# B&R Automation Studio project lab_2
Automation Studio 4.5.2.102

## Configuration lab_config

CPU 4PP065.0571-P74, AutomationRuntime D4.52, Build 4.1.2, Vc V4.52.0, Safety 1.6

### Task classes (Cpu.sw)
```
Cyclic#1 (cycle 2000 us, tolerance 0 us):
  ncsdcctrl <- ncsdcctrl.prg
Cyclic#8:
  Program1 <- Program1.prg
NcDataObjects: acp10etxen <- acp10etxen.dob, gAxis01a <- gAxis01obj.gAxis01a.dob, gAxis01i <- gAxis01obj.gAxis01i.dob, gAxis02a <- gAxis02obj.gAxis02a.dob, gAxis02i <- gAxis02obj.gAxis02i.dob
VcDataObjects: Visu <- Visu.dob
Binaries: vcpdsw, udbdef, vcrt, vcpfmtcx, Visu03, vcfile, vcgclass, arial, vcdsint, vcmgr, vcdsloc, vcfntttf, Visu02, vccovl, vcshared, arialbd, vcalarm, vcptelo, vcpdpp30, vccbtn, Visu01, vccnum, vcbclass, vcpfpp30, vctcal, TCData, iomap, asfw, Role, ashwac, sysconf, ashwd, User, arconfig, acp10cfg, Acp10map, vcctext
Libraries: Acp10man, Acp10par, NcGlobal, Acp10sdc, AsBrStr, Acp10_MC, brsystem, sys_lib, runtime, Library1, vcresman, asieccon, fileio, astime, dataobj, powerlnk
```

### Hardware
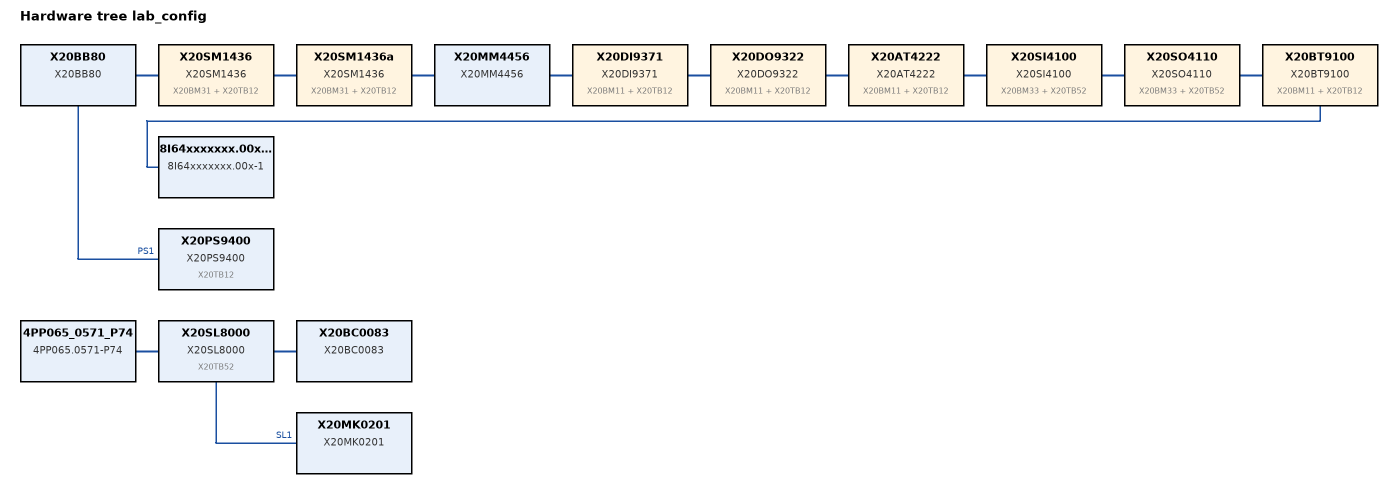
```
4PP065_0571_P74 : 4PP065.0571-P74 v1.1.2.0
  Connector IF5:
    ActivateDevice = 1
    Mode = Manual
    InternetAddress = 10.0.1.10
    SubnetMask = 255.255.255.0
  ConfigurationID = labBR
  Simulation = 1
  TimerDeviceType = EPLX2X
  TimerDevice = 4PP065_0571_P74.IF4
  TaskClassIdleTime = 2000
  Cyclic1Duration = 2000
  Cyclic1Tolerance = 0
  Cyclic1Output = 1
  VcObjectName = Visu
8I64xxxxxxx.00x-1a : 8I64xxxxxxx.00x-1 v1.3.9.1  [X2X1 -> X20BT9100.X2X1 [Cable Type=X2XCable, Length=10, Version=1.0.0.2]]
  packedETAD = packed
  packedETI = packed
  packedCMDD = packed
  packedCMI = packed
  UNS = 220
  NCR = 10
  NSP = 890
  COS = 64
  RSC = 33000
X20AT4222 : X20AT4222 v1.2.3.0  [SS1 -> X20TB12d.SS; SL -> X20BM11b.SL1]
X20BB80 : X20BB80 v1.0.2.0
X20BC0083 : X20BC0083 v2.7.0.0  [PLK1 -> X20SL8000.PLK2 [Cable Type=PowerlinkCable, Length=10, Version=1.0.0.2]; SL -> X20BB80.SL1]
X20BM11 : X20BM11 v1.0.0.1  [X2X1 -> X20MM4456.X2X2]
X20BM11a : X20BM11 v1.0.0.1  [X2X1 -> X20BM11.X2X2]
X20BM11b : X20BM11 v1.0.0.1  [X2X1 -> X20BM11a.X2X2]
X20BM11c : X20BM11 v1.0.0.1  [X2X1 -> X20BM33a.X2X2]
X20BM31 : X20BM31 v1.0.0.1  [X2X1 -> X20BB80.IF1]
X20BM31a : X20BM31 v1.0.0.1  [X2X1 -> X20BM31.X2X2]
X20BM33 : X20BM33 v1.0.0.4  [X2X1 -> X20BM11b.X2X2]
X20BM33a : X20BM33 v1.0.0.4  [X2X1 -> X20BM33.X2X2]
X20BT9100 : X20BT9100 v1.0.3.0  [SS1 -> X20TB12e.SS; SL -> X20BM11c.SL1]
X20DI9371 : X20DI9371 v1.0.2.0  [SS1 -> X20TB12b.SS; SL -> X20BM11.SL1]
X20DO9322 : X20DO9322 v1.0.3.0  [SS1 -> X20TB12c.SS; SL -> X20BM11a.SL1]
X20MK0201 : X20MK0201 v1.0.0.0  [SL -> X20SL8000.SL1]
X20MM4456 : X20MM4456 v1.1.5.0  [X2X1 -> X20BM31a.X2X2]
X20PS9400 : X20PS9400 v1.0.2.4  [SS1 -> X20TB12.SS; PS -> X20BB80.PS1]
X20SI4100 : X20SI4100 v1.10.1.1  [SS1 -> X20TB52a.SS; SL -> X20BM33.SL1]
X20SL8000 : X20SL8000 v1.6.5.1  [PLK1 -> 4PP065_0571_P74.IF4 [Cable Type=PowerlinkCable, Length=10, Version=1.0.0.2]; PLK2 -> X20BC0083.PLK1 [Cable Type=PowerlinkCable, Length=10, Version=1.0.0.2]; SS1 -> X20TB52.SS]
  SafeProject = SafeLOGIC-1
X20SM1436 : X20SM1436 v1.4.2.1  [SS1 -> X20TB12a.SS; SL -> X20BM31.SL1]
X20SM1436a : X20SM1436 v1.4.2.1  [SS1 -> X20TB12f.SS; SL -> X20BM31a.SL1]
X20SO4110 : X20SO4110 v1.10.1.1  [SS1 -> X20TB52b.SS; SL -> X20BM33a.SL1]
  SafeModuleID = 3
X20TB12 : X20TB12 v1.0.0.0
X20TB12a : X20TB12 v1.0.0.0
X20TB12b : X20TB12 v1.0.0.0
X20TB12c : X20TB12 v1.0.0.0
X20TB12d : X20TB12 v1.0.0.0
X20TB12e : X20TB12 v1.0.0.0
X20TB12f : X20TB12 v1.0.0.0
X20TB52 : X20TB52 v1.0.0.1
X20TB52a : X20TB52 v1.0.0.1
X20TB52b : X20TB52 v1.0.0.1
```

### IoMap.iom - 4PP065_0571_P74/IoMap.iom
```iecst
VAR_CONFIG
	::driveSM.STATE AT %IW."8I64xxxxxxx.00x-1a".ETAD_Input;
	::driveSM.CMD AT %QW."8I64xxxxxxx.00x-1a".CMDD_Output;
	Cyclic#1.gAxis02_DrvIf.iLifeCnt AT %IB."8I64xxxxxxx.00x-1a".SDC_LifeCnt;
	Cyclic#1.gAxis02_DrvIf.iDrvOK AT %IX."8I64xxxxxxx.00x-1a".ETAD_Input_Bool_02;
	Cyclic#1.gAxis02_DrvIf.oSetTime AT %QW."8I64xxxxxxx.00x-1a".SDC_SetTime;
	Cyclic#1.::driveSM.speed AT %QW."8I64xxxxxxx.00x-1a".LFRD_Output;
	Cyclic#1.gAxis02_DiDoIf.iLifeCntDriveReady AT %IB."8I64xxxxxxx.00x-1a".SDC_LifeCnt;
	Cyclic#1.gAxis02_DiDoIf.iLifeCntDriveEnable AT %IB."8I64xxxxxxx.00x-1a".SDC_LifeCnt;
	Cyclic#1.gAxis02_DiDoIf.oDriveEnable AT %QX."8I64xxxxxxx.00x-1a".CMDD_Output_Bool_00;
	Cyclic#1.gAxis02_ModuleOk AT %QX."8I64xxxxxxx.00x-1a".CMDD_Output_Bool_01;
	Cyclic#1.gAxis02_ModuleOk AT %QX."8I64xxxxxxx.00x-1a".CMDD_Output_Bool_02;
	Cyclic#1.gAxis02_ModuleOk AT %IX."8I64xxxxxxx.00x-1a".ModuleOk;
	Cyclic#1.gAxis02_DiDoIf.oDriveEnable AT %QX."8I64xxxxxxx.00x-1a".CMDD_Output_Bool_03;
	Cyclic#1.gAxis02_DiDoIf.iDriveReady AT %IX."8I64xxxxxxx.00x-1a".ETAD_Input_Bool_02;
	::DoorSM.direction AT %IX."X20DI9371".DigitalInput01;
	::DoorSM.s0 AT %IX."X20DI9371".DigitalInput02;
	::DoorSM.s1 AT %IX."X20DI9371".DigitalInput03;
	::DoorSM.s2 AT %IX."X20DI9371".DigitalInput04;
	::DoorSM.s3 AT %IX."X20DI9371".DigitalInput05;
	::ledSM.led1 AT %QX."X20DO9322".DigitalOutput02;
	::ledSM.led2 AT %QX."X20DO9322".DigitalOutput03;
	::ledSM.led3 AT %QX."X20DO9322".DigitalOutput04;
	::ledSM.led4 AT %QX."X20DO9322".DigitalOutput05;
END_VAR
```

### Acp10map.ncm - 4PP065_0571_P74/Motion/Acp10map.ncm
```
NcMapping (NcSwId=Acp10)
  NcObject X20SM1436_ncAXIS1 (ModuleId=X20SM1436, ModuleAddress=SDC_IF1.ST1, Type=ncAXIS, Channel=1, AcoposSimulation=Off, Disabled=TRUE, ModuleDisabled=FALSE)
  NcObject X20SM1436a_ncAXIS1 (ModuleId=X20SM1436a, ModuleAddress=SDC_IF1.ST2, Type=ncAXIS, Channel=1, AcoposSimulation=Off, Disabled=TRUE, ModuleDisabled=FALSE)
  NcObject gAxis02 (ModuleId=8I64xxxxxxx.00x-1a, ModuleAddress=SDC_IF1.ST3, Type=ncAXIS, Channel=1, AcoposSimulation=Off, InitParameter=gAxis02i, AcoposParameter=gAxis02a, Disabled=FALSE, ModuleDisabled=FALSE)
```

## Logical view

### Global.var - Global variables
```iecst
VAR
	DoorSM : DoorStateMachine;
	speed : INT := 500;
	gAxis01 : ACP10AXIS_typ;
	gAxis01_HW : SdcHwCfg_typ := (0);
	gAxis01_DrvIf : SdcDrvIf16_typ := (0);
	gAxis01_DiDoIf : SdcDiDoIf_typ := (0);
	gAxis01_ModuleOk : BOOL := 0;
	gAxis02 : ACP10AXIS_typ;
	gAxis02_HW : SdcHwCfg_typ := (0);
	gAxis02_DrvIf : SdcDrvIf16_typ := (0);
	gAxis02_DiDoIf : SdcDiDoIf_typ := (0);
	gAxis02_ModuleOk : BOOL := 0;
	ledSM : LedStateMachine;
	driveSM : DriveStateMachine;
END_VAR
```

- Visualisation Logical/Visu (not shown)

### Program Logical/Program1 (ANSIC)

#### Cyclic.c
```c
#include <bur/plctypes.h>

#ifdef _DEFAULT_INCLUDES
	#include <AsDefault.h>
#endif

void _CYCLIC ProgramCyclic(void)
{

	DoorStateMachine(&DoorSM);
	driveSM.speed = DoorSM.speed;
	DriveStateMachine(&driveSM);
	ledSM.state = DoorSM.state;
	LedStateMachine(&ledSM);
}
```

#### Init.c
```c
#include <bur/plctypes.h>

#ifdef _DEFAULT_INCLUDES
	#include <AsDefault.h>
#endif

void _INIT ProgramInit(void)
{
		driveSM.ENABLE = 1;
}
```

### Library Logical/Library1 (ANSIC)

#### Types.typ - Exported data types
```iecst
TYPE
	DoorStates :
		(
		SM_INIT,
		SM_UNKNOWN,
		SM_CLOSE,
		SM_NEG,
		SM_ACC_NEG,
		SM_DEC_NEG,
		SM_OPEN,
		SM_POS,
		SM_ACC_POS,
		SM_DEC_POS
		);
	driveCommands :
		(
		CMD_SWITCHED_ON := 7,
		CMD_DISABLE_VOLTAGE := 0,
		CMD_ENABLED := 15,
		CMD_SHUTDOWN := 6,
		STATE_READY := 33,
		STATE_DISABLED := 64,
		STATE_SWITCHED_ON := 35
		);
END_TYPE
```

#### Library1.fun - Exported functions and function blocks
```iecst
{REDUND_ERROR} FUNCTION_BLOCK LedStateMachine (*TODO: Add your comment here*) (*$GROUP=User,$CAT=User,$GROUPICON=User.png,$CATICON=User.png*)
	VAR_INPUT
		state : UINT;
	END_VAR
	VAR_OUTPUT
		led1 : BOOL;
		led2 : BOOL;
		led3 : BOOL;
		led4 : BOOL;
		timer : INT;
	END_VAR
END_FUNCTION_BLOCK

{REDUND_ERROR} FUNCTION_BLOCK DoorStateMachine (*TODO: Add your comment here*) (*$GROUP=User,$CAT=User,$GROUPICON=User.png,$CATICON=User.png*)
	VAR_INPUT
		state : UINT;
		s0 : BOOL;
		s1 : BOOL;
		s2 : BOOL;
		s3 : BOOL;
		direction : BOOL;
	END_VAR
	VAR_OUTPUT
		speed : INT;
	END_VAR
END_FUNCTION_BLOCK

{REDUND_ERROR} FUNCTION_BLOCK DriveStateMachine (*TODO: Add your comment here*) (*$GROUP=User,$CAT=User,$GROUPICON=User.png,$CATICON=User.png*)
	VAR_INPUT
		STATE : UINT;
		ENABLE : BOOL;
	END_VAR
	VAR_OUTPUT
		CMD : UINT;
		speed : INT;
	END_VAR
END_FUNCTION_BLOCK
```

#### LedStateMachine.c
```c
#include <bur/plctypes.h>
#ifdef __cplusplus
	extern "C"
	{
#endif
	#include "Library1.h"
#ifdef __cplusplus
	};
#endif
/* TODO: Add your comment here */
void LedStateMachine(struct LedStateMachine* inst)
{
	/*TODO: Add your code here*/

	switch(inst->state)
	{
		case SM_INIT:
			{

				break;
			}

		case SM_UNKNOWN:
			{
				if(inst->timer%10==0)
				{
					inst->led1=!inst->led1;
					inst->led2=!inst->led2;
					inst->led3=!inst->led3;
					inst->led4=!inst->led4;
				}
				break;
			}

		case SM_CLOSE:
			{
				inst->led1=1;
				inst->led2=1;
				inst->led3=1;
				inst->led4=1;
				break;
			}
		case SM_NEG:
			{
				inst->led1=0;
				inst->led2=0;
				inst->led3=1;
				inst->led4=1;
				break;
			}
		case SM_ACC_NEG:
			{
				inst->led1=0;
				inst->led2=0;
				inst->led3=0;
				inst->led4=1;
				break;
			}
		case SM_DEC_NEG:
			{
				inst->led1=0;
				inst->led2=1;
				inst->led3=1;
				inst->led4=1;
				break;
			}

		case SM_OPEN:
			{
				inst->led1=0;
				inst->led2=0;
				inst->led3=0;
				inst->led4=0;
				break;
			}
		case SM_POS:
			{
				inst->led1=0;
				inst->led2=0;
				inst->led3=1;
				inst->led4=1;
				break;
			}
		case SM_ACC_POS:
			{
				inst->led1=0;
				inst->led2=1;
				inst->led3=1;
				inst->led4=1;
				break;
			}
		case SM_DEC_POS:
			{
				inst->led1=0;
				inst->led2=0;
				inst->led3=0;
				inst->led4=1;
				break;
			}
	}
	inst->timer++;
}
```

#### DoorStateMachine.c
```c
#include <bur/plctypes.h>
#ifdef __cplusplus
	extern "C"
	{
#endif
	#include "Library1.h"
#ifdef __cplusplus
	};
#endif
/* TODO: Add your comment here */
void DoorStateMachine(struct DoorStateMachine* inst)
{
	/*TODO: Add your code here*/
	switch (inst->state)
	{
		case SM_INIT:
			{
				if(inst->s0==0 && inst->s1==0 && inst->s2==0 && inst->s3==0)
					inst->state=SM_UNKNOWN;
				break;
			}
		case SM_UNKNOWN:
			{
				if (inst->s0 == 1)
					inst->state=SM_CLOSE;
				if (inst->s1 == 1)
					inst->state=SM_ACC_POS;
				if (inst->s2 == 1)
					inst->state=SM_DEC_POS;
				if (inst->s3 == 1)
					inst->state=SM_OPEN;
				break;
			}
		case SM_CLOSE:
			{
				inst->speed = 0;
				if(inst->direction==1)
					inst->state=SM_ACC_POS;
				break;
			}
		case SM_ACC_NEG:
			{
				inst->speed = -200;
				if(inst->direction==1)
					inst->state=SM_DEC_POS;
				if(inst->direction==0 && inst->s2==1)
					inst->state=SM_NEG;
				break;
			}
		case SM_NEG:
			{
				inst->speed = -700;
				if(inst->direction==1)
					inst->state=SM_POS;
				if(inst->direction==0 && inst->s1==1)
					inst->state=SM_DEC_NEG;
				break;

			}

		case SM_DEC_NEG:
			{
				inst->speed = -200;
				if(inst->direction==1)
					inst->state=SM_ACC_POS;
				if(inst->direction==0 && inst->s0==1)
					inst->state=SM_CLOSE;
				break;
			}
		case SM_OPEN:
			{
				inst->speed = 0;
				if(inst->direction==0)
					inst->state=SM_ACC_NEG;
				break;
			}
		case SM_ACC_POS:
			{
				inst->speed = 200;
				if(inst->direction==0)
					inst->state=SM_DEC_NEG;
				if(inst->direction==1 && inst->s1==1)
					inst->state=SM_POS;
				break;
			}
		case SM_POS:
			{
				inst->speed = 700;
				if(inst->direction==0)
					inst->state=SM_NEG;
				if(inst->direction==1 && inst->s2==1)
					inst->state=SM_DEC_POS;
				break;
			}

		case SM_DEC_POS:
			{
				inst->speed = 200;
				if(inst->direction==0)
					inst->state=SM_ACC_NEG;
				if(inst->direction==1 && inst->s3==1)
					inst->state=SM_OPEN;

				break;
			}
	}
}
```

#### DriveStateMachine.c
```c
#include <bur/plctypes.h>
#ifdef __cplusplus
	extern "C"
	{
#endif
	#include "Library1.h"
#ifdef __cplusplus
	};
#endif
/* TODO: Add your comment here */
void DriveStateMachine(struct DriveStateMachine* inst)
{
	/*TODO: Add your code here*/
	UINT mask = inst->STATE & 0x6f;
	if(!inst->ENABLE)
	{
		inst->CMD = CMD_SHUTDOWN;
	}
	else
	{
		switch (mask)
		{
			case STATE_DISABLED:
				inst->CMD = CMD_SHUTDOWN;
				break;

			case STATE_READY:
				inst->CMD = CMD_ENABLED;
				break;

			case STATE_SWITCHED_ON:
				inst->CMD = CMD_SWITCHED_ON;
				break;
		}
	}
}
```

Listed in the project but not available here: Logical/Global.typ, Logical/Libraries, Logical/acp10etxen, Logical/ncsdcctrl, Logical/gAxis01obj, Logical/gAxis02obj, Logical/Library1/Constants.var
